(* IEC 61131-3 sources: AXOpen/src/components.rexroth.tightening/ctrl/src/TemplateComponent, 1 file *)

(* ---- TemplateComponent.st ---- *)
USING AXOpen.Core;
USING AXOpen.Messaging;
USING AXOpen.Messaging.Static;
USING AXOpen.Components.Abstractions;
USING Siemens.Simatic.S71500.Hardware.Utilities;

NAMESPACE AXOpen.Components.Rexroth.Tightening
    {S7.extern=ReadWrite}
    CLASS TemplateComponent EXTENDS AXOpen.Core.AxoComponent
        VAR PUBLIC // HEADER

        END_VAR

        VAR PUBLIC // TASKS
            {#ix-attr:[Container(Layout.Wrap)]}
            {#ix-attr:[ComponentDetails("Tasks")]}
            {#ix-set:AttributeName = "<#Restore#>"}
            RestoreTask : AXOpen.Core.AxoTask;
        END_VAR

        VAR PUBLIC // TEMPLATE TASKS
            {#ix-attr:[Container(Layout.Wrap)]}
            {#ix-attr:[ComponentDetails("Template tasks")]}
            {#ix-set:AttributeName = "<#TemplateTask_10steps_1#>"}
            TemplateTask_10steps_1 : AXOpen.Core.AxoTask;
            {#ix-attr:[Container(Layout.Wrap)]}
            {#ix-attr:[ComponentDetails("Template tasks")]}
            {#ix-set:AttributeName = "<#TemplateTask_10steps_2#>"}
            TemplateTask_10steps_2 : AXOpen.Core.AxoTask;
            {#ix-attr:[Container(Layout.Wrap)]}
            {#ix-attr:[ComponentDetails("Template tasks")]}
            {#ix-set:AttributeName = "<#TemplateTask_10steps_3#>"}
            TemplateTask_10steps_3 : AXOpen.Core.AxoTask;
            {#ix-attr:[Container(Layout.Wrap)]}
            {#ix-attr:[ComponentDetails("Template tasks")]}
            {#ix-set:AttributeName = "<#TemplateTask_10steps_4#>"}
            TemplateTask_10steps_4 : AXOpen.Core.AxoTask;
            {#ix-attr:[Container(Layout.Wrap)]}
            {#ix-attr:[ComponentDetails("Template tasks")]}
            {#ix-set:AttributeName = "<#TemplateTask_10steps_5#>"}
            TemplateTask_10steps_5 : AXOpen.Core.AxoTask;
            {#ix-attr:[Container(Layout.Wrap)]}
            {#ix-attr:[ComponentDetails("Template tasks")]}
            {#ix-set:AttributeName = "<#TemplateTask_10steps_6#>"}
            TemplateTask_10steps_6 : AXOpen.Core.AxoTask;

            {#ix-attr:[Container(Layout.Wrap)]}
            {#ix-attr:[ComponentDetails("Template tasks")]}
            {#ix-set:AttributeName = "<#TemplateTask_20steps_1#>"}
            TemplateTask_20steps_1 : AXOpen.Core.AxoTask;
            {#ix-attr:[Container(Layout.Wrap)]}
            {#ix-attr:[ComponentDetails("Template tasks")]}
            {#ix-set:AttributeName = "<#TemplateTask_20steps_2#>"}
            TemplateTask_20steps_2 : AXOpen.Core.AxoTask;
            {#ix-attr:[Container(Layout.Wrap)]}
            {#ix-attr:[ComponentDetails("Template tasks")]}
            {#ix-set:AttributeName = "<#TemplateTask_20steps_3#>"}
            TemplateTask_20steps_3 : AXOpen.Core.AxoTask;
            {#ix-attr:[Container(Layout.Wrap)]}
            {#ix-attr:[ComponentDetails("Template tasks")]}
            {#ix-set:AttributeName = "<#TemplateTask_20steps_4#>"}
            TemplateTask_20steps_4 : AXOpen.Core.AxoTask;
            {#ix-attr:[Container(Layout.Wrap)]}
            {#ix-attr:[ComponentDetails("Template tasks")]}
            {#ix-set:AttributeName = "<#TemplateTask_20steps_5#>"}
            TemplateTask_20steps_5 : AXOpen.Core.AxoTask;
            {#ix-attr:[Container(Layout.Wrap)]}
            {#ix-attr:[ComponentDetails("Template tasks")]}
            {#ix-set:AttributeName = "<#TemplateTask_20steps_6#>"}
            TemplateTask_20steps_6 : AXOpen.Core.AxoTask;

        END_VAR

        VAR PUBLIC // CONFIG
            {#ix-attr:[Container(Layout.Stack)]}
            {#ix-attr:[ComponentDetails("Config")]}
            {#ix-attr:[ReadOnly()]}
            Config  :   TemplateComponent_Config;
        END_VAR

        VAR PUBLIC // STATUS
            {#ix-attr:[Container(Layout.Stack)]}
            {#ix-attr:[ComponentDetails("Status")]}
            {#ix-attr:[ReadOnly()]}
            Status              :   TemplateComponent_Component_Status;
            Messenger           :   AXOpen.Messaging.Static.AxoMessenger;
            TaskMessenger       :   AXOpen.Messaging.Static.AxoMessenger;
        END_VAR

        VAR PUBLIC // HARDWARE SIGNALS
            {#ix-attr:[ComponentDetails("HARDWARE SIGNALS")]}
            {#ix-attr:[Container(Layout.Wrap)]}
            {#ix-attr:[Group(GroupLayout.GroupBox)]}
            {#ix-set:AttributeName = "<#Inputs#>"}
            {#ix-attr:[ReadOnly()]}
            Inputs              :  TemplateComponent_In;
            {#ix-attr:[ComponentDetails("HARDWARE SIGNALS")]}
            {#ix-attr:[Container(Layout.Wrap)]}
            {#ix-attr:[Group(GroupLayout.GroupBox)]}
            {#ix-set:AttributeName = "<#Outputs#>"}
            {#ix-attr:[ReadOnly()]}
            Outputs              :   TemplateComponent_Out;
        END_VAR

        VAR PUBLIC // HARDWARE DIAGNOSTICS TASK
            {#ix-attr:[Container(Layout.Stack)]}
            {#ix-attr:[ComponentDetails("Hardware diagnostics")]}
            {#ix-set:AttributeName = "<#Update diagnostics#>"}
            HardwareDiagnosticsTask :   AXOpen.Io.AxoHardwareDiagnostics;
        END_VAR

        VAR PRIVATE
            _hwID           :   WORD;
            _hwID_1         :   WORD;
            _hwID_2         :   WORD;
            _hwID_3         :   WORD;
            _hwID_4         :   WORD;
            _hwID_5         :   WORD;
            _hwID_6         :   WORD;
            _hwID_7         :   WORD;
            _hwID_8         :   WORD;
            _hwID_9         :   WORD;
            _hwID_10        :   WORD;
            _hwID_11        :   WORD;
            _hwID_12        :   WORD;
            _hwID_13        :   WORD;
            _hwID_14        :   WORD;
            _hwID_15        :   WORD;
            _hwID_16        :   WORD;
            _hwID_17        :   WORD;
            _hwID_18        :   WORD;
            _hwID_19        :   WORD;
            _hwID_20        :   WORD;
            _progress       :   INT;
            _infoTimer      :   AXOpen.Timers.OnDelayTimer;
            _errorTimer     :   AXOpen.Timers.OnDelayTimer;
            _returnValue    :   WORD;
            _data_in        :   ARRAY[0..254] OF BYTE;
            _data_out_1     :   ARRAY[0..0] OF BYTE;
            _data_out_2     :   ARRAY[0..1] OF BYTE;
            _data_out_4     :   ARRAY[0..3] OF BYTE;
            _data_out_8     :   ARRAY[0..7] OF BYTE;
            _data_out_255   :   ARRAY[0..254] OF BYTE;
            _word           :   WORD;
            _dword          :   DWORD;

            _initHwCheckDone        :   BOOL;
            _retval                 :   WORD;
            _geoAddr                :   GeoAddr;
            _outHwid                :   UINT;
            _startAddress           :   UDINT;
            _bytesCount             :   UINT;
        END_VAR

        ///<summary>
        /// Runs tasks and logic of this component.
        /// >[!IMPORTANT] This method must or one of its overloads be called cyclically.
        ///</summary>
        METHOD PUBLIC Run
            VAR_INPUT
                parent  : IAxoObject;
                hwID    :   WORD;
                hwID_1  :   WORD;
                hwID_2  :   WORD;
                hwID_3  :   WORD;
                hwID_4  :   WORD;
                hwID_5  :   WORD;
                hwID_6  :   WORD;
                hwID_7  :   WORD;
                hwID_8  :   WORD;
                hwID_9  :   WORD;
                hwID_10 :   WORD;
                hwID_11 :   WORD;
                hwID_12 :   WORD;
                hwID_13 :   WORD;
                hwID_14 :   WORD;
                hwID_15 :   WORD;
                hwID_16 :   WORD;
                hwID_17 :   WORD;
                hwID_18 :   WORD;
                hwID_19 :   WORD;
                hwID_20 :   WORD;
            END_VAR

            SUPER.Run(parent);

            Messenger.Serve(THIS);

            IF NOT _initHwCheckDone THEN
                IF parent = NULL THEN
                    Messenger.Activate(ULINT#700, eAxoMessageCategory#ProgrammingError);
                    Status.Error.Id := UINT#700;
                    RETURN;
                END_IF;
                IF hwID = WORD#0 THEN
                    Messenger.Activate(ULINT#701, eAxoMessageCategory#ProgrammingError);
                    Status.Error.Id := UINT#701;
                    RETURN;
                END_IF;

                _hwID                    := hwID;
                _retval := ReadSlotFromHardwareID(hardwareID := TO_UINT(_hwID), geoAddr :=_geoAddr);
                IF _retval = WORD#8090 THEN
                    Messenger.Activate(UINT#702,eAxoMessageCategory#Error);
                    Status.Error.Id := UINT#702;
                    RETURN;
                END_IF;

                //******************Slot 1*****************//
                _geoAddr.Slot   :=  UINT#1;
                _retval := ReadHardwareIDFromSlot(geoAddr := _geoAddr, hardwareID => _outHwid);
                _hwID_1 :=  TO_WORD(_outHwid);

                IF _hwID_1 = WORD#0 THEN
                    Messenger.Activate(UINT#703,eAxoMessageCategory#Error);
                    Status.Error.Id := UINT#703;
                    RETURN;
                END_IF;
                IF _retval = WORD#8091 THEN
                    Messenger.Activate(UINT#704,eAxoMessageCategory#Error);
                    Status.Error.Id := UINT#704;
                    RETURN;
                END_IF;
                IF _retval = WORD#8094 THEN
                    Messenger.Activate(UINT#705,eAxoMessageCategory#Error);
                    Status.Error.Id := UINT#705;
                    RETURN;
                END_IF;
                IF _retval = WORD#8095 THEN
                    Messenger.Activate(UINT#706,eAxoMessageCategory#Error);
                    Status.Error.Id := UINT#706;
                    RETURN;
                END_IF;
                IF _retval = WORD#8096 THEN
                    Messenger.Activate(UINT#707,eAxoMessageCategory#Error);
                    Status.Error.Id := UINT#707;
                    RETURN;
                END_IF;
                IF _retval = WORD#8097 THEN
                    Messenger.Activate(UINT#708,eAxoMessageCategory#Error);
                    Status.Error.Id := UINT#708;
                    RETURN;
                END_IF;

                //******************Slot 2*****************//
                _geoAddr.Slot   :=  UINT#2;
                _retval := ReadHardwareIDFromSlot(geoAddr := _geoAddr, hardwareID => _outHwid);
                _hwID_2 :=  TO_WORD(_outHwid);

                IF _hwID_2 = WORD#0 THEN
                    Messenger.Activate(UINT#709,eAxoMessageCategory#Error);
                    Status.Error.Id := UINT#709;
                    RETURN;
                END_IF;
                IF _retval = WORD#8091 THEN
                    Messenger.Activate(UINT#710,eAxoMessageCategory#Error);
                    Status.Error.Id := UINT#710;
                    RETURN;
                END_IF;
                IF _retval = WORD#8094 THEN
                    Messenger.Activate(UINT#711,eAxoMessageCategory#Error);
                    Status.Error.Id := UINT#711;
                    RETURN;
                END_IF;
                IF _retval = WORD#8095 THEN
                    Messenger.Activate(UINT#712,eAxoMessageCategory#Error);
                    Status.Error.Id := UINT#712;
                    RETURN;
                END_IF;
                IF _retval = WORD#8096 THEN
                    Messenger.Activate(UINT#713,eAxoMessageCategory#Error);
                    Status.Error.Id := UINT#713;
                    RETURN;
                END_IF;
                IF _retval = WORD#8097 THEN
                    Messenger.Activate(UINT#714,eAxoMessageCategory#Error);
                    Status.Error.Id := UINT#714;
                    RETURN;
                END_IF;

                //******************Slot 3*****************//
                _geoAddr.Slot   :=  UINT#3;
                _retval := ReadHardwareIDFromSlot(geoAddr := _geoAddr, hardwareID => _outHwid);
                _hwID_3 :=  TO_WORD(_outHwid);

                IF _hwID_3 = WORD#0 THEN
                    Messenger.Activate(UINT#715,eAxoMessageCategory#Error);
                    Status.Error.Id := UINT#715;
                    RETURN;
                END_IF;
                IF _retval = WORD#8091 THEN
                    Messenger.Activate(UINT#716,eAxoMessageCategory#Error);
                    Status.Error.Id := UINT#716;
                    RETURN;
                END_IF;
                IF _retval = WORD#8094 THEN
                    Messenger.Activate(UINT#717,eAxoMessageCategory#Error);
                    Status.Error.Id := UINT#717;
                    RETURN;
                END_IF;
                IF _retval = WORD#8095 THEN
                    Messenger.Activate(UINT#718,eAxoMessageCategory#Error);
                    Status.Error.Id := UINT#718;
                    RETURN;
                END_IF;
                IF _retval = WORD#8096 THEN
                    Messenger.Activate(UINT#719,eAxoMessageCategory#Error);
                    Status.Error.Id := UINT#719;
                    RETURN;
                END_IF;
                IF _retval = WORD#8097 THEN
                    Messenger.Activate(UINT#720,eAxoMessageCategory#Error);
                    Status.Error.Id := UINT#720;
                    RETURN;
                END_IF;

                //******************Slot 4*****************//
                _geoAddr.Slot   :=  UINT#4;
                _retval := ReadHardwareIDFromSlot(geoAddr := _geoAddr, hardwareID => _outHwid);
                _hwID_4 :=  TO_WORD(_outHwid);

                IF _hwID_4 = WORD#0 THEN
                    Messenger.Activate(UINT#721,eAxoMessageCategory#Error);
                    Status.Error.Id := UINT#721;
                    RETURN;
                END_IF;
                IF _retval = WORD#8091 THEN
                    Messenger.Activate(UINT#722,eAxoMessageCategory#Error);
                    Status.Error.Id := UINT#722;
                    RETURN;
                END_IF;
                IF _retval = WORD#8094 THEN
                    Messenger.Activate(UINT#723,eAxoMessageCategory#Error);
                    Status.Error.Id := UINT#723;
                    RETURN;
                END_IF;
                IF _retval = WORD#8095 THEN
                    Messenger.Activate(UINT#724,eAxoMessageCategory#Error);
                    Status.Error.Id := UINT#724;
                    RETURN;
                END_IF;
                IF _retval = WORD#8096 THEN
                    Messenger.Activate(UINT#725,eAxoMessageCategory#Error);
                    Status.Error.Id := UINT#725;
                    RETURN;
                END_IF;
                IF _retval = WORD#8097 THEN
                    Messenger.Activate(UINT#726,eAxoMessageCategory#Error);
                    Status.Error.Id := UINT#726;
                    RETURN;
                END_IF;

                //******************Slot 5*****************//
                _geoAddr.Slot   :=  UINT#5;
                _retval := ReadHardwareIDFromSlot(geoAddr := _geoAddr, hardwareID => _outHwid);
                _hwID_5 :=  TO_WORD(_outHwid);

                IF _hwID_5 = WORD#0 THEN
                    Messenger.Activate(UINT#727,eAxoMessageCategory#Error);
                    Status.Error.Id := UINT#727;
                    RETURN;
                END_IF;
                IF _retval = WORD#8091 THEN
                    Messenger.Activate(UINT#728,eAxoMessageCategory#Error);
                    Status.Error.Id := UINT#728;
                    RETURN;
                END_IF;
                IF _retval = WORD#8094 THEN
                    Messenger.Activate(UINT#729,eAxoMessageCategory#Error);
                    Status.Error.Id := UINT#729;
                    RETURN;
                END_IF;
                IF _retval = WORD#8095 THEN
                    Messenger.Activate(UINT#730,eAxoMessageCategory#Error);
                    Status.Error.Id := UINT#730;
                    RETURN;
                END_IF;
                IF _retval = WORD#8096 THEN
                    Messenger.Activate(UINT#731,eAxoMessageCategory#Error);
                    Status.Error.Id := UINT#731;
                    RETURN;
                END_IF;
                IF _retval = WORD#8097 THEN
                    Messenger.Activate(UINT#732,eAxoMessageCategory#Error);
                    Status.Error.Id := UINT#732;
                    RETURN;
                END_IF;

                //******************Slot 6*****************//
                _geoAddr.Slot   :=  UINT#6;
                _retval := ReadHardwareIDFromSlot(geoAddr := _geoAddr, hardwareID => _outHwid);
                _hwID_6 :=  TO_WORD(_outHwid);

                IF _hwID_6 = WORD#0 THEN
                    Messenger.Activate(UINT#733,eAxoMessageCategory#Error);
                    Status.Error.Id := UINT#733;
                    RETURN;
                END_IF;
                IF _retval = WORD#8091 THEN
                    Messenger.Activate(UINT#734,eAxoMessageCategory#Error);
                    Status.Error.Id := UINT#734;
                    RETURN;
                END_IF;
                IF _retval = WORD#8094 THEN
                    Messenger.Activate(UINT#735,eAxoMessageCategory#Error);
                    Status.Error.Id := UINT#735;
                    RETURN;
                END_IF;
                IF _retval = WORD#8095 THEN
                    Messenger.Activate(UINT#736,eAxoMessageCategory#Error);
                    Status.Error.Id := UINT#736;
                    RETURN;
                END_IF;
                IF _retval = WORD#8096 THEN
                    Messenger.Activate(UINT#737,eAxoMessageCategory#Error);
                    Status.Error.Id := UINT#737;
                    RETURN;
                END_IF;
                IF _retval = WORD#8097 THEN
                    Messenger.Activate(UINT#738,eAxoMessageCategory#Error);
                    Status.Error.Id := UINT#738;
                    RETURN;
                END_IF;

                //******************Slot 7*****************//
                _geoAddr.Slot   :=  UINT#7;
                _retval := ReadHardwareIDFromSlot(geoAddr := _geoAddr, hardwareID => _outHwid);
                _hwID_7 :=  TO_WORD(_outHwid);

                IF _hwID_7 = WORD#0 THEN
                    Messenger.Activate(UINT#739,eAxoMessageCategory#Error);
                    Status.Error.Id := UINT#739;
                    RETURN;
                END_IF;
                IF _retval = WORD#8091 THEN
                    Messenger.Activate(UINT#740,eAxoMessageCategory#Error);
                    Status.Error.Id := UINT#740;
                    RETURN;
                END_IF;
                IF _retval = WORD#8094 THEN
                    Messenger.Activate(UINT#741,eAxoMessageCategory#Error);
                    Status.Error.Id := UINT#741;
                    RETURN;
                END_IF;
                IF _retval = WORD#8095 THEN
                    Messenger.Activate(UINT#742,eAxoMessageCategory#Error);
                    Status.Error.Id := UINT#742;
                    RETURN;
                END_IF;
                IF _retval = WORD#8096 THEN
                    Messenger.Activate(UINT#743,eAxoMessageCategory#Error);
                    Status.Error.Id := UINT#743;
                    RETURN;
                END_IF;
                IF _retval = WORD#8097 THEN
                    Messenger.Activate(UINT#744,eAxoMessageCategory#Error);
                    Status.Error.Id := UINT#744;
                    RETURN;
                END_IF;

                //******************Slot 8*****************//
                _geoAddr.Slot   :=  UINT#8;
                _retval := ReadHardwareIDFromSlot(geoAddr := _geoAddr, hardwareID => _outHwid);
                _hwID_8 :=  TO_WORD(_outHwid);

                IF _hwID_8 = WORD#0 THEN
                    Messenger.Activate(UINT#745,eAxoMessageCategory#Error);
                    Status.Error.Id := UINT#745;
                    RETURN;
                END_IF;
                IF _retval = WORD#8091 THEN
                    Messenger.Activate(UINT#746,eAxoMessageCategory#Error);
                    Status.Error.Id := UINT#746;
                    RETURN;
                END_IF;
                IF _retval = WORD#8094 THEN
                    Messenger.Activate(UINT#747,eAxoMessageCategory#Error);
                    Status.Error.Id := UINT#747;
                    RETURN;
                END_IF;
                IF _retval = WORD#8095 THEN
                    Messenger.Activate(UINT#748,eAxoMessageCategory#Error);
                    Status.Error.Id := UINT#748;
                    RETURN;
                END_IF;
                IF _retval = WORD#8096 THEN
                    Messenger.Activate(UINT#749,eAxoMessageCategory#Error);
                    Status.Error.Id := UINT#749;
                    RETURN;
                END_IF;
                IF _retval = WORD#8097 THEN
                    Messenger.Activate(UINT#750,eAxoMessageCategory#Error);
                    Status.Error.Id := UINT#750;
                    RETURN;
                END_IF;

                //******************Slot 9*****************//
                _geoAddr.Slot   :=  UINT#9;
                _retval := ReadHardwareIDFromSlot(geoAddr := _geoAddr, hardwareID => _outHwid);
                _hwID_9 :=  TO_WORD(_outHwid);

                IF _hwID_9 = WORD#0 THEN
                    Messenger.Activate(UINT#751,eAxoMessageCategory#Error);
                    Status.Error.Id := UINT#751;
                    RETURN;
                END_IF;
                IF _retval = WORD#8091 THEN
                    Messenger.Activate(UINT#752,eAxoMessageCategory#Error);
                    Status.Error.Id := UINT#752;
                    RETURN;
                END_IF;
                IF _retval = WORD#8094 THEN
                    Messenger.Activate(UINT#753,eAxoMessageCategory#Error);
                    Status.Error.Id := UINT#753;
                    RETURN;
                END_IF;
                IF _retval = WORD#8095 THEN
                    Messenger.Activate(UINT#754,eAxoMessageCategory#Error);
                    Status.Error.Id := UINT#754;
                    RETURN;
                END_IF;
                IF _retval = WORD#8096 THEN
                    Messenger.Activate(UINT#755,eAxoMessageCategory#Error);
                    Status.Error.Id := UINT#755;
                    RETURN;
                END_IF;
                IF _retval = WORD#8097 THEN
                    Messenger.Activate(UINT#756,eAxoMessageCategory#Error);
                    Status.Error.Id := UINT#756;
                    RETURN;
                END_IF;

                //******************Slot 10*****************//
                _geoAddr.Slot   :=  UINT#10;
                _retval := ReadHardwareIDFromSlot(geoAddr := _geoAddr, hardwareID => _outHwid);
                _hwID_10 :=  TO_WORD(_outHwid);

                IF _hwID_10 = WORD#0 THEN
                    Messenger.Activate(UINT#757,eAxoMessageCategory#Error);
                    Status.Error.Id := UINT#757;
                    RETURN;
                END_IF;
                IF _retval = WORD#8091 THEN
                    Messenger.Activate(UINT#758,eAxoMessageCategory#Error);
                    Status.Error.Id := UINT#758;
                    RETURN;
                END_IF;
                IF _retval = WORD#8094 THEN
                    Messenger.Activate(UINT#759,eAxoMessageCategory#Error);
                    Status.Error.Id := UINT#759;
                    RETURN;
                END_IF;
                IF _retval = WORD#8095 THEN
                    Messenger.Activate(UINT#760,eAxoMessageCategory#Error);
                    Status.Error.Id := UINT#760;
                    RETURN;
                END_IF;
                IF _retval = WORD#8096 THEN
                    Messenger.Activate(UINT#761,eAxoMessageCategory#Error);
                    Status.Error.Id := UINT#761;
                    RETURN;
                END_IF;
                IF _retval = WORD#8097 THEN
                    Messenger.Activate(UINT#762,eAxoMessageCategory#Error);
                    Status.Error.Id := UINT#762;
                    RETURN;
                END_IF;

                //******************Slot 11*****************//
                _geoAddr.Slot   :=  UINT#11;
                _retval := ReadHardwareIDFromSlot(geoAddr := _geoAddr, hardwareID => _outHwid);
                _hwID_11 :=  TO_WORD(_outHwid);

                IF _hwID_11 = WORD#0 THEN
                    Messenger.Activate(UINT#763,eAxoMessageCategory#Error);
                    Status.Error.Id := UINT#763;
                    RETURN;
                END_IF;
                IF _retval = WORD#8091 THEN
                    Messenger.Activate(UINT#764,eAxoMessageCategory#Error);
                    Status.Error.Id := UINT#764;
                    RETURN;
                END_IF;
                IF _retval = WORD#8094 THEN
                    Messenger.Activate(UINT#765,eAxoMessageCategory#Error);
                    Status.Error.Id := UINT#765;
                    RETURN;
                END_IF;
                IF _retval = WORD#8095 THEN
                    Messenger.Activate(UINT#766,eAxoMessageCategory#Error);
                    Status.Error.Id := UINT#766;
                    RETURN;
                END_IF;
                IF _retval = WORD#8096 THEN
                    Messenger.Activate(UINT#767,eAxoMessageCategory#Error);
                    Status.Error.Id := UINT#767;
                    RETURN;
                END_IF;
                IF _retval = WORD#8097 THEN
                    Messenger.Activate(UINT#768,eAxoMessageCategory#Error);
                    Status.Error.Id := UINT#768;
                    RETURN;
                END_IF;

                //******************Slot 12*****************//
                _geoAddr.Slot   :=  UINT#12;
                _retval := ReadHardwareIDFromSlot(geoAddr := _geoAddr, hardwareID => _outHwid);
                _hwID_12 :=  TO_WORD(_outHwid);

                IF _hwID_12 = WORD#0 THEN
                    Messenger.Activate(UINT#769,eAxoMessageCategory#Error);
                    Status.Error.Id := UINT#769;
                    RETURN;
                END_IF;
                IF _retval = WORD#8091 THEN
                    Messenger.Activate(UINT#770,eAxoMessageCategory#Error);
                    Status.Error.Id := UINT#770;
                    RETURN;
                END_IF;
                IF _retval = WORD#8094 THEN
                    Messenger.Activate(UINT#771,eAxoMessageCategory#Error);
                    Status.Error.Id := UINT#771;
                    RETURN;
                END_IF;
                IF _retval = WORD#8095 THEN
                    Messenger.Activate(UINT#772,eAxoMessageCategory#Error);
                    Status.Error.Id := UINT#772;
                    RETURN;
                END_IF;
                IF _retval = WORD#8096 THEN
                    Messenger.Activate(UINT#773,eAxoMessageCategory#Error);
                    Status.Error.Id := UINT#773;
                    RETURN;
                END_IF;
                IF _retval = WORD#8097 THEN
                    Messenger.Activate(UINT#774,eAxoMessageCategory#Error);
                    Status.Error.Id := UINT#774;
                    RETURN;
                END_IF;

                //******************Slot 13*****************//
                _geoAddr.Slot   :=  UINT#13;
                _retval := ReadHardwareIDFromSlot(geoAddr := _geoAddr, hardwareID => _outHwid);
                _hwID_13 :=  TO_WORD(_outHwid);

                IF _hwID_13 = WORD#0 THEN
                    Messenger.Activate(UINT#775,eAxoMessageCategory#Error);
                    Status.Error.Id := UINT#775;
                    RETURN;
                END_IF;
                IF _retval = WORD#8091 THEN
                    Messenger.Activate(UINT#776,eAxoMessageCategory#Error);
                    Status.Error.Id := UINT#776;
                    RETURN;
                END_IF;
                IF _retval = WORD#8094 THEN
                    Messenger.Activate(UINT#777,eAxoMessageCategory#Error);
                    Status.Error.Id := UINT#777;
                    RETURN;
                END_IF;
                IF _retval = WORD#8095 THEN
                    Messenger.Activate(UINT#778,eAxoMessageCategory#Error);
                    Status.Error.Id := UINT#778;
                    RETURN;
                END_IF;
                IF _retval = WORD#8096 THEN
                    Messenger.Activate(UINT#779,eAxoMessageCategory#Error);
                    Status.Error.Id := UINT#779;
                    RETURN;
                END_IF;
                IF _retval = WORD#8097 THEN
                    Messenger.Activate(UINT#780,eAxoMessageCategory#Error);
                    Status.Error.Id := UINT#780;
                    RETURN;
                END_IF;

                //******************Slot 14*****************//
                _geoAddr.Slot   :=  UINT#14;
                _retval := ReadHardwareIDFromSlot(geoAddr := _geoAddr, hardwareID => _outHwid);
                _hwID_14 :=  TO_WORD(_outHwid);

                IF _hwID_14 = WORD#0 THEN
                    Messenger.Activate(UINT#781,eAxoMessageCategory#Error);
                    Status.Error.Id := UINT#781;
                    RETURN;
                END_IF;
                IF _retval = WORD#8091 THEN
                    Messenger.Activate(UINT#782,eAxoMessageCategory#Error);
                    Status.Error.Id := UINT#782;
                    RETURN;
                END_IF;
                IF _retval = WORD#8094 THEN
                    Messenger.Activate(UINT#783,eAxoMessageCategory#Error);
                    Status.Error.Id := UINT#783;
                    RETURN;
                END_IF;
                IF _retval = WORD#8095 THEN
                    Messenger.Activate(UINT#784,eAxoMessageCategory#Error);
                    Status.Error.Id := UINT#784;
                    RETURN;
                END_IF;
                IF _retval = WORD#8096 THEN
                    Messenger.Activate(UINT#785,eAxoMessageCategory#Error);
                    Status.Error.Id := UINT#785;
                    RETURN;
                END_IF;
                IF _retval = WORD#8097 THEN
                    Messenger.Activate(UINT#786,eAxoMessageCategory#Error);
                    Status.Error.Id := UINT#786;
                    RETURN;
                END_IF;

                //******************Slot 15*****************//
                _geoAddr.Slot   :=  UINT#15;
                _retval := ReadHardwareIDFromSlot(geoAddr := _geoAddr, hardwareID => _outHwid);
                _hwID_15 :=  TO_WORD(_outHwid);

                IF _hwID_15 = WORD#0 THEN
                    Messenger.Activate(UINT#787,eAxoMessageCategory#Error);
                    Status.Error.Id := UINT#787;
                    RETURN;
                END_IF;
                IF _retval = WORD#8091 THEN
                    Messenger.Activate(UINT#788,eAxoMessageCategory#Error);
                    Status.Error.Id := UINT#788;
                    RETURN;
                END_IF;
                IF _retval = WORD#8094 THEN
                    Messenger.Activate(UINT#789,eAxoMessageCategory#Error);
                    Status.Error.Id := UINT#789;
                    RETURN;
                END_IF;
                IF _retval = WORD#8095 THEN
                    Messenger.Activate(UINT#790,eAxoMessageCategory#Error);
                    Status.Error.Id := UINT#790;
                    RETURN;
                END_IF;
                IF _retval = WORD#8096 THEN
                    Messenger.Activate(UINT#791,eAxoMessageCategory#Error);
                    Status.Error.Id := UINT#791;
                    RETURN;
                END_IF;
                IF _retval = WORD#8097 THEN
                    Messenger.Activate(UINT#792,eAxoMessageCategory#Error);
                    Status.Error.Id := UINT#792;
                    RETURN;
                END_IF;

                //******************Slot 16*****************//
                _geoAddr.Slot   :=  UINT#16;
                _retval := ReadHardwareIDFromSlot(geoAddr := _geoAddr, hardwareID => _outHwid);
                _hwID_16 :=  TO_WORD(_outHwid);

                IF _hwID_16 = WORD#0 THEN
                    Messenger.Activate(UINT#793,eAxoMessageCategory#Error);
                    Status.Error.Id := UINT#793;
                    RETURN;
                END_IF;
                IF _retval = WORD#8091 THEN
                    Messenger.Activate(UINT#794,eAxoMessageCategory#Error);
                    Status.Error.Id := UINT#794;
                    RETURN;
                END_IF;
                IF _retval = WORD#8094 THEN
                    Messenger.Activate(UINT#795,eAxoMessageCategory#Error);
                    Status.Error.Id := UINT#795;
                    RETURN;
                END_IF;
                IF _retval = WORD#8095 THEN
                    Messenger.Activate(UINT#796,eAxoMessageCategory#Error);
                    Status.Error.Id := UINT#796;
                    RETURN;
                END_IF;
                IF _retval = WORD#8096 THEN
                    Messenger.Activate(UINT#797,eAxoMessageCategory#Error);
                    Status.Error.Id := UINT#797;
                    RETURN;
                END_IF;
                IF _retval = WORD#8097 THEN
                    Messenger.Activate(UINT#798,eAxoMessageCategory#Error);
                    Status.Error.Id := UINT#798;
                    RETURN;
                END_IF;

                //******************Slot 17*****************//
                _geoAddr.Slot   :=  UINT#17;
                _retval := ReadHardwareIDFromSlot(geoAddr := _geoAddr, hardwareID => _outHwid);
                _hwID_17 :=  TO_WORD(_outHwid);

                IF _hwID_17 = WORD#0 THEN
                    Messenger.Activate(UINT#799,eAxoMessageCategory#Error);
                    Status.Error.Id := UINT#799;
                    RETURN;
                END_IF;
                IF _retval = WORD#8091 THEN
                    Messenger.Activate(UINT#800,eAxoMessageCategory#Error);
                    Status.Error.Id := UINT#800;
                    RETURN;
                END_IF;
                IF _retval = WORD#8094 THEN
                    Messenger.Activate(UINT#801,eAxoMessageCategory#Error);
                    Status.Error.Id := UINT#801;
                    RETURN;
                END_IF;
                IF _retval = WORD#8095 THEN
                    Messenger.Activate(UINT#802,eAxoMessageCategory#Error);
                    Status.Error.Id := UINT#802;
                    RETURN;
                END_IF;
                IF _retval = WORD#8096 THEN
                    Messenger.Activate(UINT#803,eAxoMessageCategory#Error);
                    Status.Error.Id := UINT#803;
                    RETURN;
                END_IF;
                IF _retval = WORD#8097 THEN
                    Messenger.Activate(UINT#804,eAxoMessageCategory#Error);
                    Status.Error.Id := UINT#804;
                    RETURN;
                END_IF;

                //******************Slot 18*****************//
                _geoAddr.Slot   :=  UINT#18;
                _retval := ReadHardwareIDFromSlot(geoAddr := _geoAddr, hardwareID => _outHwid);
                _hwID_18 :=  TO_WORD(_outHwid);

                IF _hwID_18 = WORD#0 THEN
                    Messenger.Activate(UINT#805,eAxoMessageCategory#Error);
                    Status.Error.Id := UINT#805;
                    RETURN;
                END_IF;
                IF _retval = WORD#8091 THEN
                    Messenger.Activate(UINT#806,eAxoMessageCategory#Error);
                    Status.Error.Id := UINT#806;
                    RETURN;
                END_IF;
                IF _retval = WORD#8094 THEN
                    Messenger.Activate(UINT#807,eAxoMessageCategory#Error);
                    Status.Error.Id := UINT#807;
                    RETURN;
                END_IF;
                IF _retval = WORD#8095 THEN
                    Messenger.Activate(UINT#808,eAxoMessageCategory#Error);
                    Status.Error.Id := UINT#808;
                    RETURN;
                END_IF;
                IF _retval = WORD#8096 THEN
                    Messenger.Activate(UINT#809,eAxoMessageCategory#Error);
                    Status.Error.Id := UINT#809;
                    RETURN;
                END_IF;
                IF _retval = WORD#8097 THEN
                    Messenger.Activate(UINT#810,eAxoMessageCategory#Error);
                    Status.Error.Id := UINT#810;
                    RETURN;
                END_IF;

                //******************Slot 19*****************//
                _geoAddr.Slot   :=  UINT#19;
                _retval := ReadHardwareIDFromSlot(geoAddr := _geoAddr, hardwareID => _outHwid);
                _hwID_19 :=  TO_WORD(_outHwid);

                IF _hwID_19 = WORD#0 THEN
                    Messenger.Activate(UINT#811,eAxoMessageCategory#Error);
                    Status.Error.Id := UINT#811;
                    RETURN;
                END_IF;
                IF _retval = WORD#8091 THEN
                    Messenger.Activate(UINT#812,eAxoMessageCategory#Error);
                    Status.Error.Id := UINT#812;
                    RETURN;
                END_IF;
                IF _retval = WORD#8094 THEN
                    Messenger.Activate(UINT#813,eAxoMessageCategory#Error);
                    Status.Error.Id := UINT#813;
                    RETURN;
                END_IF;
                IF _retval = WORD#8095 THEN
                    Messenger.Activate(UINT#814,eAxoMessageCategory#Error);
                    Status.Error.Id := UINT#814;
                    RETURN;
                END_IF;
                IF _retval = WORD#8096 THEN
                    Messenger.Activate(UINT#815,eAxoMessageCategory#Error);
                    Status.Error.Id := UINT#815;
                    RETURN;
                END_IF;
                IF _retval = WORD#8097 THEN
                    Messenger.Activate(UINT#816,eAxoMessageCategory#Error);
                    Status.Error.Id := UINT#816;
                    RETURN;
                END_IF;

                //******************Slot 20*****************//
                _geoAddr.Slot   :=  UINT#20;
                _retval := ReadHardwareIDFromSlot(geoAddr := _geoAddr, hardwareID => _outHwid);
                _hwID_20 :=  TO_WORD(_outHwid);

                IF _hwID_20 = WORD#0 THEN
                    Messenger.Activate(UINT#817,eAxoMessageCategory#Error);
                    Status.Error.Id := UINT#817;
                    RETURN;
                END_IF;
                IF _retval = WORD#8091 THEN
                    Messenger.Activate(UINT#818,eAxoMessageCategory#Error);
                    Status.Error.Id := UINT#818;
                    RETURN;
                END_IF;
                IF _retval = WORD#8094 THEN
                    Messenger.Activate(UINT#819,eAxoMessageCategory#Error);
                    Status.Error.Id := UINT#819;
                    RETURN;
                END_IF;
                IF _retval = WORD#8095 THEN
                    Messenger.Activate(UINT#820,eAxoMessageCategory#Error);
                    Status.Error.Id := UINT#820;
                    RETURN;
                END_IF;
                IF _retval = WORD#8096 THEN
                    Messenger.Activate(UINT#821,eAxoMessageCategory#Error);
                    Status.Error.Id := UINT#821;
                    RETURN;
                END_IF;
                IF _retval = WORD#8097 THEN
                    Messenger.Activate(UINT#822,eAxoMessageCategory#Error);
                    Status.Error.Id := UINT#822;
                    RETURN;
                END_IF;

                _hwID       :=  hwID;
                _hwID_1     :=  hwID_1;
                _hwID_2     :=  hwID_2;
                _hwID_3     :=  hwID_3;
                _hwID_4     :=  hwID_4;
                _hwID_5     :=  hwID_5;
                _hwID_6     :=  hwID_6;
                _hwID_7     :=  hwID_7;
                _hwID_8     :=  hwID_8;
                _hwID_9     :=  hwID_9;
                _hwID_10    :=  hwID_10;
                _hwID_11    :=  hwID_11;
                _hwID_12    :=  hwID_12;
                _hwID_13    :=  hwID_13;
                _hwID_14    :=  hwID_14;
                _hwID_15    :=  hwID_15;
                _hwID_16    :=  hwID_16;
                _hwID_17    :=  hwID_17;
                _hwID_18    :=  hwID_18;
                _hwID_19    :=  hwID_19;
                _hwID_20    :=  hwID_20;

                IF parent = NULL THEN
                    Messenger.Activate(UINT#830,eAxoMessageCategory#Error);
                    Status.Error.Id := UINT#830;
                    RETURN;
                END_IF;

                IF _hwID  = WORD#0 THEN
                    Messenger.Activate(UINT#831,eAxoMessageCategory#Error);
                    Status.Error.Id := UINT#831;
                    RETURN;
                END_IF;

                IF _hwID_1  = WORD#0 THEN
                    Messenger.Activate(UINT#832,eAxoMessageCategory#Error);
                    Status.Error.Id := UINT#832;
                    RETURN;
                END_IF;

                IF _hwID_2  = WORD#0 THEN
                    Messenger.Activate(UINT#833,eAxoMessageCategory#Error);
                    Status.Error.Id := UINT#833;
                    RETURN;
                END_IF;

                IF _hwID_3  = WORD#0 THEN
                    Messenger.Activate(UINT#834,eAxoMessageCategory#Error);
                    Status.Error.Id := UINT#834;
                    RETURN;
                END_IF;

                IF _hwID_4  = WORD#0 THEN
                    Messenger.Activate(UINT#835,eAxoMessageCategory#Error);
                    Status.Error.Id := UINT#835;
                    RETURN;
                END_IF;

                IF _hwID_5  = WORD#0 THEN
                    Messenger.Activate(UINT#836,eAxoMessageCategory#Error);
                    Status.Error.Id := UINT#836;
                    RETURN;
                END_IF;

                IF _hwID_6  = WORD#0 THEN
                    Messenger.Activate(UINT#837,eAxoMessageCategory#Error);
                    Status.Error.Id := UINT#837;
                    RETURN;
                END_IF;

                IF _hwID_7  = WORD#0 THEN
                    Messenger.Activate(UINT#838,eAxoMessageCategory#Error);
                    Status.Error.Id := UINT#838;
                    RETURN;
                END_IF;

                IF _hwID_8  = WORD#0 THEN
                    Messenger.Activate(UINT#839,eAxoMessageCategory#Error);
                    Status.Error.Id := UINT#839;
                    RETURN;
                END_IF;

                IF _hwID_9  = WORD#0 THEN
                    Messenger.Activate(UINT#840,eAxoMessageCategory#Error);
                    Status.Error.Id := UINT#840;
                    RETURN;
                END_IF;

                IF _hwID_10  = WORD#0 THEN
                    Messenger.Activate(UINT#841,eAxoMessageCategory#Error);
                    Status.Error.Id := UINT#841;
                    RETURN;
                END_IF;

                IF _hwID_11  = WORD#0 THEN
                    Messenger.Activate(UINT#842,eAxoMessageCategory#Error);
                    Status.Error.Id := UINT#842;
                    RETURN;
                END_IF;

                IF _hwID_12  = WORD#0 THEN
                    Messenger.Activate(UINT#843,eAxoMessageCategory#Error);
                    Status.Error.Id := UINT#843;
                    RETURN;
                END_IF;

                IF _hwID_13  = WORD#0 THEN
                    Messenger.Activate(UINT#844,eAxoMessageCategory#Error);
                    Status.Error.Id := UINT#844;
                    RETURN;
                END_IF;

                IF _hwID_14  = WORD#0 THEN
                    Messenger.Activate(UINT#845,eAxoMessageCategory#Error);
                    Status.Error.Id := UINT#845;
                    RETURN;
                END_IF;

                IF _hwID_15  = WORD#0 THEN
                    Messenger.Activate(UINT#846,eAxoMessageCategory#Error);
                    Status.Error.Id := UINT#846;
                    RETURN;
                END_IF;

                IF _hwID_16  = WORD#0 THEN
                    Messenger.Activate(UINT#847,eAxoMessageCategory#Error);
                    Status.Error.Id := UINT#847;
                    RETURN;
                END_IF;

                IF _hwID_17  = WORD#0 THEN
                    Messenger.Activate(UINT#848,eAxoMessageCategory#Error);
                    Status.Error.Id := UINT#848;
                    RETURN;
                END_IF;

                IF _hwID_18  = WORD#0 THEN
                    Messenger.Activate(UINT#849,eAxoMessageCategory#Error);
                    Status.Error.Id := UINT#849;
                    RETURN;
                END_IF;

                IF _hwID_19  = WORD#0 THEN
                    Messenger.Activate(UINT#850,eAxoMessageCategory#Error);
                    Status.Error.Id := UINT#850;
                    RETURN;
                END_IF;

                IF _hwID_20  = WORD#0 THEN
                    Messenger.Activate(UINT#851,eAxoMessageCategory#Error);
                    Status.Error.Id := UINT#851;
                    RETURN;
                END_IF;

                _initHwCheckDone    := TRUE;
            END_IF;

            //***********Update inputs **************

            _returnValue := Siemens.Simatic.S71500.DistributedIO.ReadData(_hwID_1 ,_data_in);
            IF _returnValue > WORD#0 THEN
                Messenger.Activate(UINT#861, eAxoMessageCategory#ProgrammingError);
                Status.Error.Id := UINT#861;
                RETURN;
            END_IF;

            // TemplateComponentInputStructure_hwID_1.Item1  :=      _data_in[0].%X0;
            // TemplateComponentInputStructure_hwID_1.Item2  :=      _data_in[0].%X1;
            // TemplateComponentInputStructure_hwID_1.Item3  :=      _data_in[0].%X2;
            // TemplateComponentInputStructure_hwID_1.Item4  :=      _data_in[0].%X3;
            // TemplateComponentInputStructure_hwID_1.Item5  :=      _data_in[0].%X4;

            _returnValue := Siemens.Simatic.S71500.DistributedIO.ReadData(_hwID_2 ,_data_in);
            IF _returnValue > WORD#0 THEN
                Messenger.Activate(UINT#862, eAxoMessageCategory#ProgrammingError);
                Status.Error.Id := UINT#862;
                RETURN;
            END_IF;

            // TemplateComponentInputStructure_hwID_2.Item1  :=      _data_in[0].%X0;
            // TemplateComponentInputStructure_hwID_2.Item2  :=      _data_in[0].%X1;
            // TemplateComponentInputStructure_hwID_2.Item3  :=      _data_in[0].%X2;
            // TemplateComponentInputStructure_hwID_2.Item4  :=      _data_in[0].%X3;
            // TemplateComponentInputStructure_hwID_2.Item5  :=      _data_in[0].%X4;

            _returnValue := Siemens.Simatic.S71500.DistributedIO.ReadData(_hwID_3 ,_data_in);
            IF _returnValue > WORD#0 THEN
                Messenger.Activate(UINT#863, eAxoMessageCategory#ProgrammingError);
                Status.Error.Id := UINT#863;
                RETURN;
            END_IF;

            // TemplateComponentInputStructure_hwID_3.Item1  :=      _data_in[0].%X0;
            // TemplateComponentInputStructure_hwID_3.Item2  :=      _data_in[0].%X1;
            // TemplateComponentInputStructure_hwID_3.Item3  :=      _data_in[0].%X2;
            // TemplateComponentInputStructure_hwID_3.Item4  :=      _data_in[0].%X3;
            // TemplateComponentInputStructure_hwID_3.Item5  :=      _data_in[0].%X4;

            _returnValue := Siemens.Simatic.S71500.DistributedIO.ReadData(_hwID_4 ,_data_in);
            IF _returnValue > WORD#0 THEN
                Messenger.Activate(UINT#864, eAxoMessageCategory#ProgrammingError);
                Status.Error.Id := UINT#864;
                RETURN;
            END_IF;

            // TemplateComponentInputStructure_hwID_4.Item1  :=      _data_in[0].%X0;
            // TemplateComponentInputStructure_hwID_4.Item2  :=      _data_in[0].%X1;
            // TemplateComponentInputStructure_hwID_4.Item3  :=      _data_in[0].%X2;
            // TemplateComponentInputStructure_hwID_4.Item4  :=      _data_in[0].%X3;
            // TemplateComponentInputStructure_hwID_4.Item5  :=      _data_in[0].%X4;

            _returnValue := Siemens.Simatic.S71500.DistributedIO.ReadData(_hwID_5 ,_data_in);
            IF _returnValue > WORD#0 THEN
                Messenger.Activate(UINT#865, eAxoMessageCategory#ProgrammingError);
                Status.Error.Id := UINT#865;
                RETURN;
            END_IF;

            // TemplateComponentInputStructure_hwID_5.Item1  :=      _data_in[0].%X0;
            // TemplateComponentInputStructure_hwID_5.Item2  :=      _data_in[0].%X1;
            // TemplateComponentInputStructure_hwID_5.Item3  :=      _data_in[0].%X2;
            // TemplateComponentInputStructure_hwID_5.Item4  :=      _data_in[0].%X3;
            // TemplateComponentInputStructure_hwID_5.Item5  :=      _data_in[0].%X4;

            _returnValue := Siemens.Simatic.S71500.DistributedIO.ReadData(_hwID_6 ,_data_in);
            IF _returnValue > WORD#0 THEN
                Messenger.Activate(UINT#866, eAxoMessageCategory#ProgrammingError);
                Status.Error.Id := UINT#866;
                RETURN;
            END_IF;

            // _word.%B1                                                           :=  _data_in[0];
            // _word.%B0                                                           :=  _data_in[1];
            // TemplateComponentInputStructure_hwID_6.Item1                        :=  TO_UINT(_word);
            // _word.%B1                                                           :=  _data_in[2];
            // _word.%B0                                                           :=  _data_in[3];
            // TemplateComponentInputStructure_hwID_6.Item2                        :=  TO_UINT(_word);
            // _word.%B1                                                           :=  _data_in[4];
            // _word.%B0                                                           :=  _data_in[5];
            // TemplateComponentInputStructure_hwID_6.Item3                        :=  TO_UINT(_word);
            // _word.%B1                                                           :=  _data_in[6];
            // _word.%B0                                                           :=  _data_in[7];
            // TemplateComponentInputStructure_hwID_6.Item4                        :=  TO_UINT(_word);

            _returnValue := Siemens.Simatic.S71500.DistributedIO.ReadData(_hwID_7 ,_data_in);
            IF _returnValue > WORD#0 THEN
                Messenger.Activate(UINT#867, eAxoMessageCategory#ProgrammingError);
                Status.Error.Id := UINT#867;
                RETURN;
            END_IF;

            // _dword.%B3                                                          :=  _data_in[0];
            // _dword.%B2                                                          :=  _data_in[1];
            // _dword.%B1                                                          :=  _data_in[2];
            // _dword.%B0                                                          :=  _data_in[3];
            // TemplateComponentInputStructure_hwID_7.Item1                        :=  TO_DINT(_dword);
            // _dword.%B3                                                          :=  _data_in[4];
            // _dword.%B2                                                          :=  _data_in[5];
            // _dword.%B1                                                          :=  _data_in[6];
            // _dword.%B0                                                          :=  _data_in[7];
            // TemplateComponentInputStructure_hwID_7.Item2                        :=  TO_REAL(_dword);

            _returnValue := Siemens.Simatic.S71500.DistributedIO.ReadData(_hwID_8 ,_data_in);
            IF _returnValue > WORD#0 THEN
                Messenger.Activate(UINT#868, eAxoMessageCategory#ProgrammingError);
                Status.Error.Id := UINT#868;
                RETURN;
            END_IF;

            // _dword.%B3                                                          :=  _data_in[0];
            // _dword.%B2                                                          :=  _data_in[1];
            // _dword.%B1                                                          :=  _data_in[2];
            // _dword.%B0                                                          :=  _data_in[3];
            // TemplateComponentInputStructure_hwID_8.Item1                        :=  TO_DINT(_dword);
            // _dword.%B3                                                          :=  _data_in[4];
            // _dword.%B2                                                          :=  _data_in[5];
            // _dword.%B1                                                          :=  _data_in[6];
            // _dword.%B0                                                          :=  _data_in[7];
            // TemplateComponentInputStructure_hwID_8.Item2                        :=  TO_REAL(_dword);

            _returnValue := Siemens.Simatic.S71500.DistributedIO.ReadData(_hwID_9 ,_data_in);
            IF _returnValue > WORD#0 THEN
                Messenger.Activate(UINT#869, eAxoMessageCategory#ProgrammingError);
                Status.Error.Id := UINT#869;
                RETURN;
            END_IF;

            // _dword.%B3                                                          :=  _data_in[0];
            // _dword.%B2                                                          :=  _data_in[1];
            // _dword.%B1                                                          :=  _data_in[2];
            // _dword.%B0                                                          :=  _data_in[3];
            // TemplateComponentInputStructure_hwID_9.Item1                        :=  TO_DINT(_dword);
            // _dword.%B3                                                          :=  _data_in[4];
            // _dword.%B2                                                          :=  _data_in[5];
            // _dword.%B1                                                          :=  _data_in[6];
            // _dword.%B0                                                          :=  _data_in[7];
            // TemplateComponentInputStructure_hwID_9.Item2                        :=  TO_REAL(_dword);

            _returnValue := Siemens.Simatic.S71500.DistributedIO.ReadData(_hwID_10 ,_data_in);
            IF _returnValue > WORD#0 THEN
                Messenger.Activate(UINT#870, eAxoMessageCategory#ProgrammingError);
                Status.Error.Id := UINT#870;
                RETURN;
            END_IF;

            // _dword.%B3                                                          :=  _data_in[0];
            // _dword.%B2                                                          :=  _data_in[1];
            // _dword.%B1                                                          :=  _data_in[2];
            // _dword.%B0                                                          :=  _data_in[3];
            // TemplateComponentInputStructure_hwID_10.Item1                        :=  TO_DINT(_dword);
            // _dword.%B3                                                          :=  _data_in[4];
            // _dword.%B2                                                          :=  _data_in[5];
            // _dword.%B1                                                          :=  _data_in[6];
            // _dword.%B0                                                          :=  _data_in[7];
            // TemplateComponentInputStructure_hwID_10.Item2                        :=  TO_REAL(_dword);

            //*************INITIALIZATION*************
            RestoreTask.Run(THIS);
            TemplateTask_10steps_1.Run(THIS);
            TemplateTask_10steps_2.Run(THIS);
            TemplateTask_10steps_3.Run(THIS);
            TemplateTask_10steps_4.Run(THIS);
            TemplateTask_10steps_5.Run(THIS);
            TemplateTask_10steps_6.Run(THIS);
            TemplateTask_20steps_1.Run(THIS);
            TemplateTask_20steps_2.Run(THIS);
            TemplateTask_20steps_3.Run(THIS);
            TemplateTask_20steps_4.Run(THIS);
            TemplateTask_20steps_5.Run(THIS);
            TemplateTask_20steps_6.Run(THIS);

            //****************************************

            //********************Diagnostics*********
            HardwareDiagnosticsTask.Run(THIS,_hwID);
            //****************************************

            //*************RESTORE********************
            RestoreTask.IsDisabled := FALSE;
            IF RestoreTask.Execute(THIS) THEN
                THIS.Restore();
            END_IF;
            //****************************************

            //*************TemplateTask_10steps_1**************
            TemplateTask_10steps_1.SetIsDisabled(FALSE);
            IF TemplateTask_10steps_1.StartTriggered() THEN
                Status.Action.Id :=  UINT#100;
            END_IF;
            Messenger.ActivateOnCondition(ULINT#100,TemplateTask_10steps_1.IsBusy(), eAxoMessageCategory#Info);
            Messenger.ActivateOnCondition(ULINT#101,TemplateTask_10steps_1.IsDone(), eAxoMessageCategory#Info);
            IF TemplateTask_10steps_1.Execute(THIS) THEN
                IF _progress = 0 THEN
                    Status.Error.Id := UINT#0;
                    TaskMessenger.Restore();
                    THIS.CallTimers(FALSE);
                    _progress := 300;
                END_IF;

                IF _progress = 300 THEN                                                                                     // TemplateTask_10steps_1 running: , <add the detailed description of the current action 1>
                    TaskMessenger.ActivateOnCondition(ULINT#500, _infoTimer.output, eAxoMessageCategory#Warning);
                    IF _infoTimer.output THEN
                        Status.Error.Id := UINT#500;
                    END_IF;

                    IF TRUE THEN
                        THIS.CallTimers(FALSE);
                        _progress := 301;
                    END_IF;
                END_IF;

                IF _progress = 301 THEN                                                                                     // TemplateTask_10steps_1 running: , <add the detailed description of the current action 2>
                    TaskMessenger.ActivateOnCondition(ULINT#501, _infoTimer.output, eAxoMessageCategory#Warning);
                    IF _infoTimer.output THEN
                        Status.Error.Id := UINT#501;
                    END_IF;

                    IF TRUE THEN
                        THIS.CallTimers(FALSE);
                        _progress := 302;
                    END_IF;
                END_IF;

                IF _progress = 302 THEN                                                                                     // TemplateTask_10steps_1 running: , <add the detailed description of the current action 3>
                    TaskMessenger.ActivateOnCondition(ULINT#502, _infoTimer.output, eAxoMessageCategory#Warning);
                    IF _infoTimer.output THEN
                        Status.Error.Id := UINT#502;
                    END_IF;

                    IF TRUE THEN
                        THIS.CallTimers(FALSE);
                        _progress := 303;
                    END_IF;
                END_IF;

                IF _progress = 303 THEN                                                                                     // TemplateTask_10steps_1 running: , <add the detailed description of the current action 4>
                    TaskMessenger.ActivateOnCondition(ULINT#503, _infoTimer.output, eAxoMessageCategory#Warning);
                    IF _infoTimer.output THEN
                        Status.Error.Id := UINT#503;
                    END_IF;

                    IF TRUE THEN
                        THIS.CallTimers(FALSE);
                        _progress := 304;
                    END_IF;
                END_IF;

                IF _progress = 304 THEN                                                                                     // TemplateTask_10steps_1 running: , <add the detailed description of the current action 5>
                    TaskMessenger.ActivateOnCondition(ULINT#504, _infoTimer.output, eAxoMessageCategory#Warning);
                    IF _infoTimer.output THEN
                        Status.Error.Id := UINT#504;
                    END_IF;

                    IF TRUE THEN
                        THIS.CallTimers(FALSE);
                        _progress := 305;
                    END_IF;
                END_IF;

                IF _progress = 305 THEN                                                                                     // TemplateTask_10steps_1 running: , <add the detailed description of the current action 6>
                    TaskMessenger.ActivateOnCondition(ULINT#505, _infoTimer.output, eAxoMessageCategory#Warning);
                    IF _infoTimer.output THEN
                        Status.Error.Id := UINT#505;
                    END_IF;

                    IF TRUE THEN
                        THIS.CallTimers(FALSE);
                        _progress := 306;
                    END_IF;
                END_IF;

                IF _progress = 306 THEN                                                                                     // TemplateTask_10steps_1 running: , <add the detailed description of the current action 7>
                    TaskMessenger.ActivateOnCondition(ULINT#506, _infoTimer.output, eAxoMessageCategory#Warning);
                    IF _infoTimer.output THEN
                        Status.Error.Id := UINT#506;
                    END_IF;

                    IF TRUE THEN
                        THIS.CallTimers(FALSE);
                        _progress := 307;
                    END_IF;
                END_IF;

                IF _progress = 307 THEN                                                                                     // TemplateTask_10steps_1 running: , <add the detailed description of the current action 8>
                    TaskMessenger.ActivateOnCondition(ULINT#507, _infoTimer.output, eAxoMessageCategory#Warning);
                    IF _infoTimer.output THEN
                        Status.Error.Id := UINT#507;
                    END_IF;

                    IF TRUE THEN
                        THIS.CallTimers(FALSE);
                        _progress := 308;
                    END_IF;
                END_IF;

                IF _progress = 308 THEN                                                                                     // TemplateTask_10steps_1 running: , <add the detailed description of the current action 9>
                    TaskMessenger.ActivateOnCondition(ULINT#508, _infoTimer.output, eAxoMessageCategory#Warning);
                    IF _infoTimer.output THEN
                        Status.Error.Id := UINT#508;
                    END_IF;

                    IF TRUE THEN
                        THIS.CallTimers(FALSE);
                        _progress := 309;
                    END_IF;
                END_IF;

                IF _progress = 309 THEN                                                                                     // TemplateTask_10steps_1 running: , <add the detailed description of the current action 10>
                    TemplateTask_10steps_1.DoneWhen(TRUE);
                END_IF;

                THIS.CallTimers(TRUE);

                TemplateTask_10steps_1.ThrowWhen(_errorTimer.output);
                Status.Action.Id := TO_UINT(_progress);
                TemplateTask_10steps_1.ThrowWhen(TemplateTask_10steps_1.Duration >= Config.ErrorTime ,'TemplateTask_10steps_1 error.');
            END_IF;
            IF TemplateTask_10steps_1.DoneReached() THEN
                Status.Action.Id :=  UINT#101;
                Status.Error.Id :=  UINT#0;
            ELSIF TemplateTask_10steps_1.ErrorOccured() THEN
                Status.Action.Id :=  UINT#900;
                Status.Error.Id  :=  UINT#900;
            ELSIF TemplateTask_10steps_1.AbortTriggered()THEN
                Status.Action.Id :=  UINT#901;
                Status.Error.Id  :=  UINT#901;
            END_IF;
            Messenger.ActivateOnCondition(ULINT#900,TemplateTask_10steps_1.HasError(), eAxoMessageCategory#Error);
            Messenger.ActivateOnCondition(ULINT#901,TemplateTask_10steps_1.IsAborted(), eAxoMessageCategory#Error);
            Messenger.ActivateOnCondition(ULINT#102,TemplateTask_10steps_1.RestoreTriggered() , eAxoMessageCategory#Error);
            IF TemplateTask_10steps_1.RestoreTriggered() AND _progress >= 300 AND _progress <= 309  THEN
                Status.Action.Id :=  UINT#102;
                _progress := 0;
            END_IF;
            //**************************************************

            //*************TemplateTask_10steps_2***************
            TemplateTask_10steps_2.SetIsDisabled(FALSE);
            IF TemplateTask_10steps_2.StartTriggered() THEN
                Status.Action.Id :=  UINT#110;
            END_IF;
            Messenger.ActivateOnCondition(ULINT#110,TemplateTask_10steps_2.IsBusy(), eAxoMessageCategory#Info);
            Messenger.ActivateOnCondition(ULINT#111,TemplateTask_10steps_2.IsDone(), eAxoMessageCategory#Info);
            IF TemplateTask_10steps_2.Execute(THIS) THEN
                IF _progress = 0 THEN
                    Status.Error.Id := UINT#0;
                    TaskMessenger.Restore();
                    THIS.CallTimers(FALSE);
                    _progress := 310;
                END_IF;

                IF _progress = 310 THEN                                                                                     // TemplateTask_10steps_2 running: , <add the detailed description of the current action 1>
                    TaskMessenger.ActivateOnCondition(ULINT#510, _infoTimer.output, eAxoMessageCategory#Warning);
                    IF _infoTimer.output THEN
                        Status.Error.Id := UINT#510;
                    END_IF;

                    IF TRUE THEN
                        THIS.CallTimers(FALSE);
                        _progress := 311;
                    END_IF;
                END_IF;

                IF _progress = 311 THEN                                                                                     // TemplateTask_10steps_2 running: , <add the detailed description of the current action 2>
                    TaskMessenger.ActivateOnCondition(ULINT#511, _infoTimer.output, eAxoMessageCategory#Warning);
                    IF _infoTimer.output THEN
                        Status.Error.Id := UINT#511;
                    END_IF;

                    IF TRUE THEN
                        THIS.CallTimers(FALSE);
                        _progress := 312;
                    END_IF;
                END_IF;

                IF _progress = 312 THEN                                                                                     // TemplateTask_10steps_2 running: , <add the detailed description of the current action 3>
                    TaskMessenger.ActivateOnCondition(ULINT#512, _infoTimer.output, eAxoMessageCategory#Warning);
                    IF _infoTimer.output THEN
                        Status.Error.Id := UINT#512;
                    END_IF;

                    IF TRUE THEN
                        THIS.CallTimers(FALSE);
                        _progress := 313;
                    END_IF;
                END_IF;

                IF _progress = 313 THEN                                                                                     // TemplateTask_10steps_2 running: , <add the detailed description of the current action 4>
                    TaskMessenger.ActivateOnCondition(ULINT#513, _infoTimer.output, eAxoMessageCategory#Warning);
                    IF _infoTimer.output THEN
                        Status.Error.Id := UINT#513;
                    END_IF;

                    IF TRUE THEN
                        THIS.CallTimers(FALSE);
                        _progress := 314;
                    END_IF;
                END_IF;

                IF _progress = 314 THEN                                                                                     // TemplateTask_10steps_2 running: , <add the detailed description of the current action 5>
                    TaskMessenger.ActivateOnCondition(ULINT#514, _infoTimer.output, eAxoMessageCategory#Warning);
                    IF _infoTimer.output THEN
                        Status.Error.Id := UINT#514;
                    END_IF;

                    IF TRUE THEN
                        THIS.CallTimers(FALSE);
                        _progress := 315;
                    END_IF;
                END_IF;

                IF _progress = 315 THEN                                                                                     // TemplateTask_10steps_2 running: , <add the detailed description of the current action 6>
                    TaskMessenger.ActivateOnCondition(ULINT#515, _infoTimer.output, eAxoMessageCategory#Warning);
                    IF _infoTimer.output THEN
                        Status.Error.Id := UINT#515;
                    END_IF;

                    IF TRUE THEN
                        THIS.CallTimers(FALSE);
                        _progress := 316;
                    END_IF;
                END_IF;

                IF _progress = 316 THEN                                                                                     // TemplateTask_10steps_2 running: , <add the detailed description of the current action 7>
                    TaskMessenger.ActivateOnCondition(ULINT#516, _infoTimer.output, eAxoMessageCategory#Warning);
                    IF _infoTimer.output THEN
                        Status.Error.Id := UINT#516;
                    END_IF;

                    IF TRUE THEN
                        THIS.CallTimers(FALSE);
                        _progress := 317;
                    END_IF;
                END_IF;

                IF _progress = 317 THEN                                                                                     // TemplateTask_10steps_2 running: , <add the detailed description of the current action 8>
                    TaskMessenger.ActivateOnCondition(ULINT#517, _infoTimer.output, eAxoMessageCategory#Warning);
                    IF _infoTimer.output THEN
                        Status.Error.Id := UINT#517;
                    END_IF;

                    IF TRUE THEN
                        THIS.CallTimers(FALSE);
                        _progress := 318;
                    END_IF;
                END_IF;

                IF _progress = 318 THEN                                                                                     // TemplateTask_10steps_2 running: , <add the detailed description of the current action 9>
                    TaskMessenger.ActivateOnCondition(ULINT#518, _infoTimer.output, eAxoMessageCategory#Warning);
                    IF _infoTimer.output THEN
                        Status.Error.Id := UINT#518;
                    END_IF;

                    IF TRUE THEN
                        THIS.CallTimers(FALSE);
                        _progress := 319;
                    END_IF;
                END_IF;

                IF _progress = 319 THEN                                                                                     // TemplateTask_10steps_2 running: , <add the detailed description of the current action 10>
                    TemplateTask_10steps_2.DoneWhen(TRUE);
                END_IF;

                THIS.CallTimers(TRUE);

                TemplateTask_10steps_2.ThrowWhen(_errorTimer.output);
                Status.Action.Id := TO_UINT(_progress);
                TemplateTask_10steps_2.ThrowWhen(TemplateTask_10steps_2.Duration >= Config.ErrorTime ,'TemplateTask_10steps_2 error.');
            END_IF;
            IF TemplateTask_10steps_2.DoneReached() THEN
                Status.Action.Id :=  UINT#111;
                Status.Error.Id :=  UINT#0;
            ELSIF TemplateTask_10steps_2.ErrorOccured() THEN
                Status.Action.Id :=  UINT#910;
                Status.Error.Id  :=  UINT#910;
            ELSIF TemplateTask_10steps_2.AbortTriggered()THEN
                Status.Action.Id :=  UINT#911;
                Status.Error.Id  :=  UINT#911;
            END_IF;
            Messenger.ActivateOnCondition(ULINT#910,TemplateTask_10steps_2.HasError(), eAxoMessageCategory#Error);
            Messenger.ActivateOnCondition(ULINT#911,TemplateTask_10steps_2.IsAborted(), eAxoMessageCategory#Error);
            Messenger.ActivateOnCondition(ULINT#112,TemplateTask_10steps_2.RestoreTriggered() , eAxoMessageCategory#Error);
            IF TemplateTask_10steps_2.RestoreTriggered() AND _progress >= 310 AND _progress <= 319  THEN
                Status.Action.Id :=  UINT#112;
                _progress := 0;
            END_IF;
            //**************************************************

            //*************TemplateTask_10steps_3***************
            TemplateTask_10steps_3.SetIsDisabled(FALSE);
            IF TemplateTask_10steps_3.StartTriggered() THEN
                Status.Action.Id :=  UINT#120;
            END_IF;
            Messenger.ActivateOnCondition(ULINT#120,TemplateTask_10steps_3.IsBusy(), eAxoMessageCategory#Info);
            Messenger.ActivateOnCondition(ULINT#121,TemplateTask_10steps_3.IsDone(), eAxoMessageCategory#Info);
            IF TemplateTask_10steps_3.Execute(THIS) THEN
                IF _progress = 0 THEN
                    Status.Error.Id := UINT#0;
                    TaskMessenger.Restore();
                    THIS.CallTimers(FALSE);
                    _progress := 320;
                END_IF;

                IF _progress = 320 THEN                                                                                     // TemplateTask_10steps_3 running: , <add the detailed description of the current action 1>
                    TaskMessenger.ActivateOnCondition(ULINT#520, _infoTimer.output, eAxoMessageCategory#Warning);
                    IF _infoTimer.output THEN
                        Status.Error.Id := UINT#520;
                    END_IF;

                    IF TRUE THEN
                        THIS.CallTimers(FALSE);
                        _progress := 321;
                    END_IF;
                END_IF;

                IF _progress = 321 THEN                                                                                     // TemplateTask_10steps_3 running: , <add the detailed description of the current action 2>
                    TaskMessenger.ActivateOnCondition(ULINT#521, _infoTimer.output, eAxoMessageCategory#Warning);
                    IF _infoTimer.output THEN
                        Status.Error.Id := UINT#521;
                    END_IF;

                    IF TRUE THEN
                        THIS.CallTimers(FALSE);
                        _progress := 322;
                    END_IF;
                END_IF;

                IF _progress = 322 THEN                                                                                     // TemplateTask_10steps_3 running: , <add the detailed description of the current action 3>
                    TaskMessenger.ActivateOnCondition(ULINT#522, _infoTimer.output, eAxoMessageCategory#Warning);
                    IF _infoTimer.output THEN
                        Status.Error.Id := UINT#522;
                    END_IF;

                    IF TRUE THEN
                        THIS.CallTimers(FALSE);
                        _progress := 323;
                    END_IF;
                END_IF;

                IF _progress = 323 THEN                                                                                     // TemplateTask_10steps_3 running: , <add the detailed description of the current action 4>
                    TaskMessenger.ActivateOnCondition(ULINT#523, _infoTimer.output, eAxoMessageCategory#Warning);
                    IF _infoTimer.output THEN
                        Status.Error.Id := UINT#523;
                    END_IF;

                    IF TRUE THEN
                        THIS.CallTimers(FALSE);
                        _progress := 324;
                    END_IF;
                END_IF;

                IF _progress = 324 THEN                                                                                     // TemplateTask_10steps_3 running: , <add the detailed description of the current action 5>
                    TaskMessenger.ActivateOnCondition(ULINT#524, _infoTimer.output, eAxoMessageCategory#Warning);
                    IF _infoTimer.output THEN
                        Status.Error.Id := UINT#524;
                    END_IF;

                    IF TRUE THEN
                        THIS.CallTimers(FALSE);
                        _progress := 325;
                    END_IF;
                END_IF;

                IF _progress = 325 THEN                                                                                     // TemplateTask_10steps_3 running: , <add the detailed description of the current action 6>
                    TaskMessenger.ActivateOnCondition(ULINT#525, _infoTimer.output, eAxoMessageCategory#Warning);
                    IF _infoTimer.output THEN
                        Status.Error.Id := UINT#525;
                    END_IF;

                    IF TRUE THEN
                        THIS.CallTimers(FALSE);
                        _progress := 326;
                    END_IF;
                END_IF;

                IF _progress = 326 THEN                                                                                     // TemplateTask_10steps_3 running: , <add the detailed description of the current action 7>
                    TaskMessenger.ActivateOnCondition(ULINT#526, _infoTimer.output, eAxoMessageCategory#Warning);
                    IF _infoTimer.output THEN
                        Status.Error.Id := UINT#526;
                    END_IF;

                    IF TRUE THEN
                        THIS.CallTimers(FALSE);
                        _progress := 327;
                    END_IF;
                END_IF;

                IF _progress = 327 THEN                                                                                     // TemplateTask_10steps_3 running: , <add the detailed description of the current action 8>
                    TaskMessenger.ActivateOnCondition(ULINT#527, _infoTimer.output, eAxoMessageCategory#Warning);
                    IF _infoTimer.output THEN
                        Status.Error.Id := UINT#527;
                    END_IF;

                    IF TRUE THEN
                        THIS.CallTimers(FALSE);
                        _progress := 328;
                    END_IF;
                END_IF;

                IF _progress = 328 THEN                                                                                     // TemplateTask_10steps_3 running: , <add the detailed description of the current action 9>
                    TaskMessenger.ActivateOnCondition(ULINT#528, _infoTimer.output, eAxoMessageCategory#Warning);
                    IF _infoTimer.output THEN
                        Status.Error.Id := UINT#528;
                    END_IF;

                    IF TRUE THEN
                        THIS.CallTimers(FALSE);
                        _progress := 329;
                    END_IF;
                END_IF;

                IF _progress = 329 THEN                                                                                     // TemplateTask_10steps_3 running: , <add the detailed description of the current action 10>
                    TemplateTask_10steps_3.DoneWhen(TRUE);
                END_IF;

                THIS.CallTimers(TRUE);

                TemplateTask_10steps_3.ThrowWhen(_errorTimer.output);
                Status.Action.Id := TO_UINT(_progress);
                TemplateTask_10steps_3.ThrowWhen(TemplateTask_10steps_3.Duration >= Config.ErrorTime ,'TemplateTask_10steps_3 error.');
            END_IF;
            IF TemplateTask_10steps_3.DoneReached() THEN
                Status.Action.Id :=  UINT#121;
                Status.Error.Id :=  UINT#0;
            ELSIF TemplateTask_10steps_3.ErrorOccured() THEN
                Status.Action.Id :=  UINT#920;
                Status.Error.Id  :=  UINT#920;
            ELSIF TemplateTask_10steps_3.AbortTriggered()THEN
                Status.Action.Id :=  UINT#921;
                Status.Error.Id  :=  UINT#921;
            END_IF;
            Messenger.ActivateOnCondition(ULINT#920,TemplateTask_10steps_3.HasError(), eAxoMessageCategory#Error);
            Messenger.ActivateOnCondition(ULINT#921,TemplateTask_10steps_3.IsAborted(), eAxoMessageCategory#Error);
            Messenger.ActivateOnCondition(ULINT#122,TemplateTask_10steps_3.RestoreTriggered() , eAxoMessageCategory#Error);
            IF TemplateTask_10steps_3.RestoreTriggered() AND _progress >= 320 AND _progress <= 329  THEN
                Status.Action.Id :=  UINT#122;
                _progress := 0;
            END_IF;
            //**************************************************

            //*************TemplateTask_10steps_4***************
            TemplateTask_10steps_4.SetIsDisabled(FALSE);
            IF TemplateTask_10steps_4.StartTriggered() THEN
                Status.Action.Id :=  UINT#130;
            END_IF;
            Messenger.ActivateOnCondition(ULINT#130,TemplateTask_10steps_4.IsBusy(), eAxoMessageCategory#Info);
            Messenger.ActivateOnCondition(ULINT#131,TemplateTask_10steps_4.IsDone(), eAxoMessageCategory#Info);
            IF TemplateTask_10steps_4.Execute(THIS) THEN
                IF _progress = 0 THEN
                    Status.Error.Id := UINT#0;
                    TaskMessenger.Restore();
                    THIS.CallTimers(FALSE);
                    _progress := 330;
                END_IF;

                IF _progress = 330 THEN                                                                                     // TemplateTask_10steps_4 running: , <add the detailed description of the current action 1>
                    TaskMessenger.ActivateOnCondition(ULINT#530, _infoTimer.output, eAxoMessageCategory#Warning);
                    IF _infoTimer.output THEN
                        Status.Error.Id := UINT#530;
                    END_IF;

                    IF TRUE THEN
                        THIS.CallTimers(FALSE);
                        _progress := 331;
                    END_IF;
                END_IF;

                IF _progress = 331 THEN                                                                                     // TemplateTask_10steps_4 running: , <add the detailed description of the current action 2>
                    TaskMessenger.ActivateOnCondition(ULINT#531, _infoTimer.output, eAxoMessageCategory#Warning);
                    IF _infoTimer.output THEN
                        Status.Error.Id := UINT#531;
                    END_IF;

                    IF TRUE THEN
                        THIS.CallTimers(FALSE);
                        _progress := 332;
                    END_IF;
                END_IF;

                IF _progress = 332 THEN                                                                                     // TemplateTask_10steps_4 running: , <add the detailed description of the current action 3>
                    TaskMessenger.ActivateOnCondition(ULINT#532, _infoTimer.output, eAxoMessageCategory#Warning);
                    IF _infoTimer.output THEN
                        Status.Error.Id := UINT#532;
                    END_IF;

                    IF TRUE THEN
                        THIS.CallTimers(FALSE);
                        _progress := 333;
                    END_IF;
                END_IF;

                IF _progress = 333 THEN                                                                                     // TemplateTask_10steps_4 running: , <add the detailed description of the current action 4>
                    TaskMessenger.ActivateOnCondition(ULINT#533, _infoTimer.output, eAxoMessageCategory#Warning);
                    IF _infoTimer.output THEN
                        Status.Error.Id := UINT#533;
                    END_IF;

                    IF TRUE THEN
                        THIS.CallTimers(FALSE);
                        _progress := 334;
                    END_IF;
                END_IF;

                IF _progress = 334 THEN                                                                                     // TemplateTask_10steps_4 running: , <add the detailed description of the current action 5>
                    TaskMessenger.ActivateOnCondition(ULINT#534, _infoTimer.output, eAxoMessageCategory#Warning);
                    IF _infoTimer.output THEN
                        Status.Error.Id := UINT#534;
                    END_IF;

                    IF TRUE THEN
                        THIS.CallTimers(FALSE);
                        _progress := 335;
                    END_IF;
                END_IF;

                IF _progress = 335 THEN                                                                                     // TemplateTask_10steps_4 running: , <add the detailed description of the current action 6>
                    TaskMessenger.ActivateOnCondition(ULINT#535, _infoTimer.output, eAxoMessageCategory#Warning);
                    IF _infoTimer.output THEN
                        Status.Error.Id := UINT#535;
                    END_IF;

                    IF TRUE THEN
                        THIS.CallTimers(FALSE);
                        _progress := 336;
                    END_IF;
                END_IF;

                IF _progress = 336 THEN                                                                                     // TemplateTask_10steps_4 running: , <add the detailed description of the current action 7>
                    TaskMessenger.ActivateOnCondition(ULINT#536, _infoTimer.output, eAxoMessageCategory#Warning);
                    IF _infoTimer.output THEN
                        Status.Error.Id := UINT#536;
                    END_IF;

                    IF TRUE THEN
                        THIS.CallTimers(FALSE);
                        _progress := 337;
                    END_IF;
                END_IF;

                IF _progress = 337 THEN                                                                                     // TemplateTask_10steps_4 running: , <add the detailed description of the current action 8>
                    TaskMessenger.ActivateOnCondition(ULINT#537, _infoTimer.output, eAxoMessageCategory#Warning);
                    IF _infoTimer.output THEN
                        Status.Error.Id := UINT#537;
                    END_IF;

                    IF TRUE THEN
                        THIS.CallTimers(FALSE);
                        _progress := 338;
                    END_IF;
                END_IF;

                IF _progress = 338 THEN                                                                                     // TemplateTask_10steps_4 running: , <add the detailed description of the current action 9>
                    TaskMessenger.ActivateOnCondition(ULINT#538, _infoTimer.output, eAxoMessageCategory#Warning);
                    IF _infoTimer.output THEN
                        Status.Error.Id := UINT#538;
                    END_IF;

                    IF TRUE THEN
                        THIS.CallTimers(FALSE);
                        _progress := 339;
                    END_IF;
                END_IF;

                IF _progress = 339 THEN                                                                                     // TemplateTask_10steps_4 running: , <add the detailed description of the current action 10>
                    TemplateTask_10steps_4.DoneWhen(TRUE);
                END_IF;

                THIS.CallTimers(TRUE);

                TemplateTask_10steps_4.ThrowWhen(_errorTimer.output);
                Status.Action.Id := TO_UINT(_progress);
                TemplateTask_10steps_4.ThrowWhen(TemplateTask_10steps_4.Duration >= Config.ErrorTime ,'TemplateTask_10steps_4 error.');
            END_IF;
            IF TemplateTask_10steps_4.DoneReached() THEN
                Status.Action.Id :=  UINT#131;
                Status.Error.Id :=  UINT#0;
            ELSIF TemplateTask_10steps_4.ErrorOccured() THEN
                Status.Action.Id :=  UINT#930;
                Status.Error.Id  :=  UINT#930;
            ELSIF TemplateTask_10steps_4.AbortTriggered()THEN
                Status.Action.Id :=  UINT#931;
                Status.Error.Id  :=  UINT#931;
            END_IF;
            Messenger.ActivateOnCondition(ULINT#930,TemplateTask_10steps_4.HasError(), eAxoMessageCategory#Error);
            Messenger.ActivateOnCondition(ULINT#931,TemplateTask_10steps_4.IsAborted(), eAxoMessageCategory#Error);
            Messenger.ActivateOnCondition(ULINT#132,TemplateTask_10steps_4.RestoreTriggered() , eAxoMessageCategory#Error);
            IF TemplateTask_10steps_4.RestoreTriggered() AND _progress >= 330 AND _progress <= 339  THEN
                Status.Action.Id :=  UINT#132;
                _progress := 0;
            END_IF;
            //**************************************************

            //*************TemplateTask_10steps_5***************
            TemplateTask_10steps_5.SetIsDisabled(FALSE);
            IF TemplateTask_10steps_5.StartTriggered() THEN
                Status.Action.Id :=  UINT#140;
            END_IF;
            Messenger.ActivateOnCondition(ULINT#140,TemplateTask_10steps_5.IsBusy(), eAxoMessageCategory#Info);
            Messenger.ActivateOnCondition(ULINT#141,TemplateTask_10steps_5.IsDone(), eAxoMessageCategory#Info);
            IF TemplateTask_10steps_5.Execute(THIS) THEN
                IF _progress = 0 THEN
                    Status.Error.Id := UINT#0;
                    TaskMessenger.Restore();
                    THIS.CallTimers(FALSE);
                    _progress := 340;
                END_IF;

                IF _progress = 340 THEN                                                                                     // TemplateTask_10steps_5 running: , <add the detailed description of the current action 1>
                    TaskMessenger.ActivateOnCondition(ULINT#540, _infoTimer.output, eAxoMessageCategory#Warning);
                    IF _infoTimer.output THEN
                        Status.Error.Id := UINT#540;
                    END_IF;

                    IF TRUE THEN
                        THIS.CallTimers(FALSE);
                        _progress := 341;
                    END_IF;
                END_IF;

                IF _progress = 341 THEN                                                                                     // TemplateTask_10steps_5 running: , <add the detailed description of the current action 2>
                    TaskMessenger.ActivateOnCondition(ULINT#541, _infoTimer.output, eAxoMessageCategory#Warning);
                    IF _infoTimer.output THEN
                        Status.Error.Id := UINT#541;
                    END_IF;

                    IF TRUE THEN
                        THIS.CallTimers(FALSE);
                        _progress := 342;
                    END_IF;
                END_IF;

                IF _progress = 342 THEN                                                                                     // TemplateTask_10steps_5 running: , <add the detailed description of the current action 3>
                    TaskMessenger.ActivateOnCondition(ULINT#542, _infoTimer.output, eAxoMessageCategory#Warning);
                    IF _infoTimer.output THEN
                        Status.Error.Id := UINT#542;
                    END_IF;

                    IF TRUE THEN
                        THIS.CallTimers(FALSE);
                        _progress := 343;
                    END_IF;
                END_IF;

                IF _progress = 343 THEN                                                                                     // TemplateTask_10steps_5 running: , <add the detailed description of the current action 4>
                    TaskMessenger.ActivateOnCondition(ULINT#544, _infoTimer.output, eAxoMessageCategory#Warning);
                    IF _infoTimer.output THEN
                        Status.Error.Id := UINT#544;
                    END_IF;

                    IF TRUE THEN
                        THIS.CallTimers(FALSE);
                        _progress := 344;
                    END_IF;
                END_IF;

                IF _progress = 344 THEN                                                                                     // TemplateTask_10steps_5 running: , <add the detailed description of the current action 5>
                    TaskMessenger.ActivateOnCondition(ULINT#544, _infoTimer.output, eAxoMessageCategory#Warning);
                    IF _infoTimer.output THEN
                        Status.Error.Id := UINT#544;
                    END_IF;

                    IF TRUE THEN
                        THIS.CallTimers(FALSE);
                        _progress := 345;
                    END_IF;
                END_IF;

                IF _progress = 345 THEN                                                                                     // TemplateTask_10steps_5 running: , <add the detailed description of the current action 6>
                    TaskMessenger.ActivateOnCondition(ULINT#545, _infoTimer.output, eAxoMessageCategory#Warning);
                    IF _infoTimer.output THEN
                        Status.Error.Id := UINT#545;
                    END_IF;
